{attribute 'GeneratedUsingTerminal: EL3182-0000-0016'}
{attribute addProperty BoxType "EL3182-0000-0016"}
{attribute addProperty Id "Ch_2_Al_InputsCh_2_Al_Inputs_4794C08310"}
{attribute addProperty CRC "3654104786"}
{attribute addProperty Size "10"}
TYPE Ch_2_D9CD36D2 :
STRUCT
	{attribute addProperty Name "Ch_2_Al_Inputs"}
	Ch_2_Al_Inputs  : Ch_2_Al_Inputs_4794C083;
END_STRUCT
END_TYPE

(* stored: Version 1.2.0.0, ProductVersion 3.1.4024.9
   DUT Ch_2_D9CD36D2: Id {1f9f2972-2375-4737-af2d-6f39de09a3b7} *)
